(* IEC 61131-3 sources: Industry-PLC-LLM/data/PLCBEAD_repo/PLCBEAD_PLCEmbed-main/PLC-BEAD/Source/GEB/UTC_TO_LTIME, 1 file *)

(* ---- UTC_TO_LTIME.ST ---- *)
FUNCTION _INT_TO_UDINT:UDINT
	VAR_INPUT
		IN :	INT;
	END_VAR

	_INT_TO_UDINT := DINT_TO_UDINT(INT_TO_DINT(IN));
END_FUNCTION

FUNCTION DT_TO_DATE2:UDINT
	VAR_INPUT
		IN :	UDINT;
	END_VAR

	DT_TO_DATE2 := (IN / UDINT#86400) * UDINT#86400;
END_FUNCTION

FUNCTION YEAR_OF_DATE:INT
	VAR_INPUT
		IDATE :	UDINT;
	END_VAR

	YEAR_OF_DATE := UDINT_TO_INT((IDATE+UDINT#43200) / UDINT#31557600 + UDINT#1970);
END_FUNCTION

FUNCTION SET_DT:UDINT

	VAR_INPUT
		YEAR  : INT;
		MONTH :	INT;
		DAY  : INT;
		HOUR : INT;
		MINUTE : INT;
		SECOND : INT;
	END_VAR

	SET_DT := SET_DATE(YEAR, MONTH, DAY) + _INT_TO_UDINT(SECOND) + _INT_TO_UDINT(MINUTE) * UDINT#60 + _INT_TO_UDINT(HOUR) * UDINT#3600;

END_FUNCTION

FUNCTION SET_DATE:UDINT

	VAR_INPUT
		YEAR  :	INT;
		MONTH :	INT;
		DAY  :	INT;
	END_VAR

	VAR
		count :	INT;
	END_VAR

	IF MONTH > 2 THEN
		count := (MONTH - 1) * 30;
		IF MONTH > 7 THEN
			count := count + DWORD_TO_INT(SHR(DINT_TO_DWORD(INT_TO_DINT(MONTH) - INT_TO_DINT(3)),1));
		ELSE
			count := count + DWORD_TO_INT(SHR(DINT_TO_DWORD(INT_TO_DINT(MONTH) - INT_TO_DINT(4)),1));
		END_IF;
		IF SHL(INT_TO_WORD(YEAR),14) = WORD#0 THEN
			count := count + 1;
		END_IF;
	ELSE
		count := (MONTH - 1) * 31;
	END_IF;
	SET_DATE := (_INT_TO_UDINT(count + DAY  - 1) + DWORD_TO_UDINT(SHR(UDINT_TO_DWORD(_INT_TO_UDINT(YEAR) * UDINT#1461 - UDINT#2878169), 2))) * UDINT#86400;

END_FUNCTION

FUNCTION DST:BOOL
	VAR_INPUT
		UTC :	UDINT;
	END_VAR

	VAR
		yr :	INT;
		yr4 :	UDINT;
		ltc :	UDINT;
		IDATE :	UDINT;
	END_VAR

	yr := YEAR_OF_DATE(DT_TO_DATE2(UTC));
	ltc := UTC;
	IDATE := SET_DT(yr, 3, 31, 1, 0, 0);
	yr4 := DWORD_TO_UDINT(SHR(INT_TO_DWORD(5 * yr), 2)) + UDINT#1;
	DST := (IDATE - ((yr4 + UDINT#3) MOD UDINT#7) * UDINT#86400 <= ltc) AND (IDATE + (UDINT#214 - (yr4) MOD UDINT#7) * UDINT#86400 > ltc);

END_FUNCTION

FUNCTION UTC_TO_LTIME:UDINT

	VAR_INPUT
		UTC :	UDINT;
		DST_ENABLE :	BOOL;
		TIME_ZONE_OFFSET :	INT;
	END_VAR

	VAR
		tmp :	INT;
	END_VAR

	UTC_TO_LTIME := UTC + _INT_TO_UDINT(TIME_ZONE_OFFSET) * UDINT#60 + BOOL_TO_UDINT(DST_ENABLE AND DST(UTC)) * UDINT#3600;

	tmp := TIME_ZONE_OFFSET * 60 + BOOL_TO_INT(DST_ENABLE AND DST(UTC)) * 3600;
	IF tmp < 0 THEN
		UTC_TO_LTIME := UTC - _INT_TO_UDINT(ABS(tmp));
	ELSE
		UTC_TO_LTIME := UTC + _INT_TO_UDINT(tmp);
	END_IF;

END_FUNCTION

PROGRAM program0
  VAR
	UTC :	UDINT;
	DST_ENABLE :	BOOL;
	TIME_ZONE_OFFSET :	INT;
    CEIL5_OUT : UDINT;
  END_VAR

  CEIL5_OUT := UTC_TO_LTIME(UTC, DST_ENABLE, TIME_ZONE_OFFSET);
END_PROGRAM
